(* PLC project Project1, 未知 未命名 1 *)
(* stored: creationDateTime 2018-01-05T00:28:37, modificationDateTime 2018-01-14T18:44:09 *)

TYPE datatype0 : REAL := 1.0;
END_TYPE

TYPE datatype1 : STRUCT
  pp : DINT;
  qq : DINT;
END_STRUCT;
END_TYPE

PROGRAM program0
  VAR
    LocalVar0 : DINT;
  END_VAR
  VAR_INPUT
    input1 : BOOL;
  END_VAR
  VAR_OUTPUT
    output2 : BOOL;
  END_VAR
  VAR_IN_OUT
    inout : REAL;
  END_VAR

            I am ychj；；
 She is cdj
          
END_PROGRAM

PROGRAM program1
  VAR
    LocalVar0 : DINT;
  END_VAR
  VAR_INPUT
    input2 : DINT;
  END_VAR
  VAR_OUTPUT
    output3 : DINT;
  END_VAR
  VAR_IN_OUT
    inout : DINT;
  END_VAR

            LocalVar0 := -1;
output3 := input2;

          
END_PROGRAM

FUNCTION fun0 : REAL
  VAR_INPUT RETAIN
    var1 : REAL := 8.0;
  END_VAR

            LocalVar0 := 2;
output := LocalVar0;
          
END_FUNCTION

FUNCTION_BLOCK FB0
  VAR
    LocalVar0 : DINT;
  END_VAR
  VAR_OUTPUT
    output2 : DINT;
  END_VAR

            LocalVar0 := 0;
output2 := LocalVar0;
          
END_FUNCTION_BLOCK

CONFIGURATION config
  RESOURCE resource1 ON PLC
    VAR_GLOBAL RETAIN
      globalVar : BOOL := True;
    END_VAR
    TASK task0(INTERVAL := T#20ms, PRIORITY := 0);
    PROGRAM instance0 WITH task0 : program0;
  END_RESOURCE
  RESOURCE resource0 ON PLC
    VAR_GLOBAL
      LocalVar0 : DINT;
      LocalVar1 : BOOL;
    END_VAR
    TASK task1(SINGLE := LocalVar1, PRIORITY := 7);
    TASK task2(INTERVAL := T#8ms, PRIORITY := 4);
    PROGRAM inst WITH task1 : program1;
    PROGRAM pg2 : program0;
  END_RESOURCE
END_CONFIGURATION
